{attribute 'obsolete' := 'Use E_PnuematicActuatorPositionState'}
TYPE ENUM_PnuematicActuatorPositionState : E_PnuematicActuatorPositionState; END_TYPE

(* stored: Version 1.1.0.1
   DUT ENUM_PnuematicActuatorPositionState: Id {96d1580c-0314-463d-8f39-3ba2700ff149} *)
